# EPICS alarm handler configuration: mps_database/bare/alarms/areas/mpln_bc2b_mp03.alhConfig
GROUP NULL MPLN:BC2B:MP03:1
$ALIAS MPS Link Node 66
$GUIDANCE
LTUH MPS
   Group Name: MPLN:BC2B:MP03:1
   Summary PV:  MPLN:BC2B:MP03:1:STATSUMY
$END
CHANNEL  MPLN:BC2B:MP03:1    MPLN:BC2B:MP03:1:MPS_EN_RBV		-----
CHANNEL  MPLN:BC2B:MP03:1    MPLN:BC2B:MP03:1:LC1_MODE_RBV		-----
